{attribute 'qualified_only'}
{attribute 'strict'}
TYPE E_StateSortingAutoCylinder :
(
	DetectBox := 0,
	CylToWork,
	CylToBase
);
END_TYPE

(* stored: Version 1.1.0.1, ProductVersion 3.1.4024.2
   DUT E_StateSortingAutoCylinder: Id {65f2f8a0-5a1e-4570-872f-969d2bcf55aa} *)
